Fanuc KAREL source: kt00266.KL

-- PROVISIONAL review KL for V1013-1; original PC SHA256 341149ea9d016813ffe26b1f3e98905fe3961286b15a88fcbd48db17042d9240
-- Incomplete behavior may be omitted. Consult companion uncertainty JSON. Do not deploy.
PROGRAM KT00266
%NOLOCKGROUP
VAR
  S1 : STRING[80]
  S2 : STRING[80]
  OUT : BOOLEAN
BEGIN
  -- UNRESOLVED_PC offsets 5-14; opcodes 3F,75
  -- UNRESOLVED_PC offsets 19-28; opcodes 3F,75
  -- UNRESOLVED_PC offsets 33-42; opcodes 3F,75
  -- UNRESOLVED_PC offsets 47-56; opcodes 3F,75
  -- UNRESOLVED_PC offsets 61-80; opcodes 73,73,83,23
  -- UNRESOLVED_PC offsets 85-89; opcodes 7F
END KT00266
